INTERFACE ITF_Control1_HMI_Connector_Command EXTENDS ITF_BaseControlElement_HMI_Connector_Command

END_INTERFACE

(* stored: Version 1.1.0.1
   Itf ITF_Control1_HMI_Connector_Command: Id {b817769b-9bc0-013c-1e6e-21f6f58930f2} *)
